SUBAPPLICATION tastend_TON_5s (* Subapplication Type *)
  (* Standard: 61499-2; Description: Copyright (c) 2024 Meisterschulen am Ostbahnhof This program and the accompanying materials are made available under the terms of the Eclipse Public License 2.0 which is available at https://www.eclipse.org/legal/epl-2.0/ SPDX-License-Identifier: EPL-2.0 *)
  (* Version 1.0, 2024-10-23, Franz Höpfinger, Meisterschulen am Ostbahnhof *)
  PACKAGE Uebungen::sys;
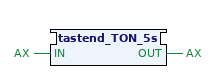
  SOCKETS
    IN : adapter::types::unidirectional::AX;
  END_SOCKETS
  PLUGS
    OUT : adapter::types::unidirectional::AX;
  END_PLUGS
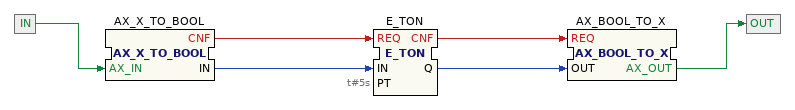
  FBS
    AX_X_TO_BOOL : adapter::conversion::unidirectional::AX_X_TO_BOOL;
    AX_BOOL_TO_X : adapter::conversion::unidirectional::AX_BOOL_TO_X;
    E_TON : iec61499::events::timers::E_TON(PT := t#5s);
  END_FBS
  EVENT_CONNECTIONS
    AX_X_TO_BOOL.CNF TO E_TON.REQ;
    E_TON.CNF TO AX_BOOL_TO_X.REQ;
  END_CONNECTIONS
  DATA_CONNECTIONS
    E_TON.Q TO AX_BOOL_TO_X.OUT;
    AX_X_TO_BOOL.IN TO E_TON.IN;
  END_CONNECTIONS
  ADAPTER_CONNECTIONS
    IN TO AX_X_TO_BOOL.AX_IN;
    AX_BOOL_TO_X.AX_OUT TO OUT;
  END_CONNECTIONS
END_SUBAPPLICATION
